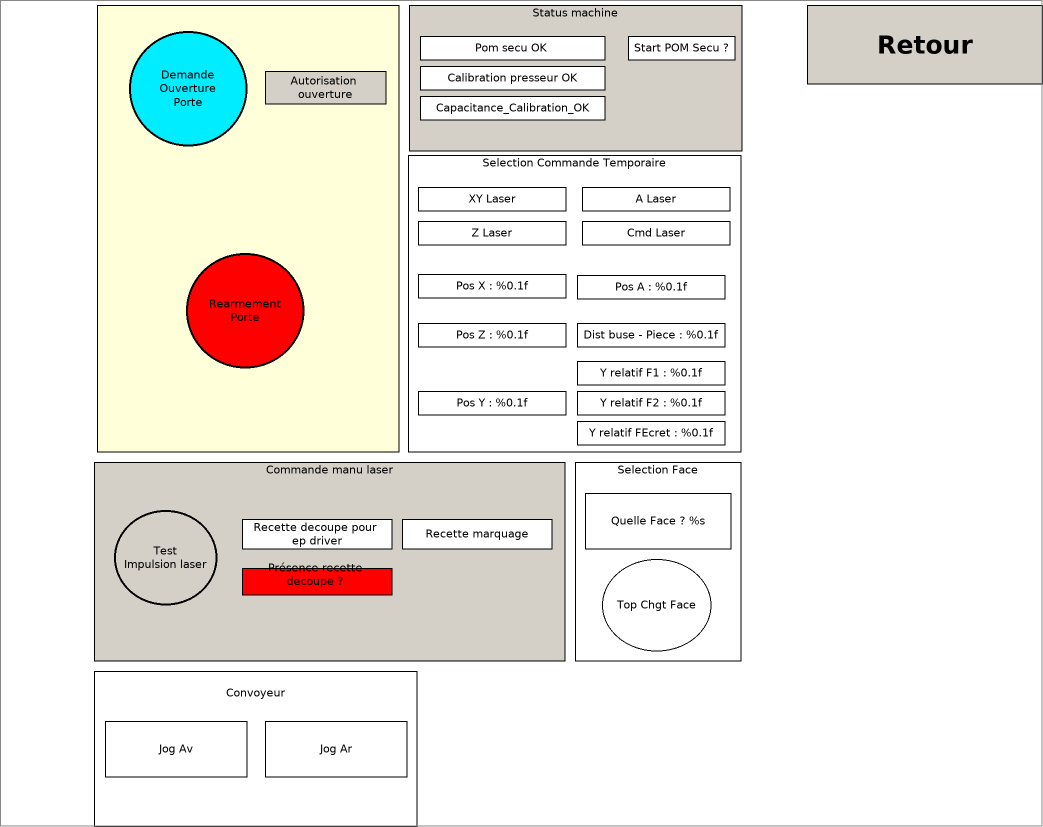
VISUALIZATION Porte_secu  // 1043x827
    Rectangle (94,462 471x199), "Commande manu laser"
    Rectangle (94,671 323x156), "Convoyeur"
        tap Gestion_ConvLaser.Jog_Av_ConvLaser
    Rectangle (97,5 302x447)
    Ellipse (129,31 118x115), "Demande Ouverture Porte", colour toggle: Attente_Arret_Propre and Clignotant_t_lent
        tap Global_Laser.Dmd_VerrDeverr_Porte
    Ellipse (186,253 118x115), "Rearmement Porte", colour toggle: RAZ_Pnoz_PorteLaser
        tap Global_Laser.Bp_Raz_Pnoz_Laser
    Rectangle (807,5 236x79), "Retour"
        OnMouseClick: change screen: Selection_Rep
        OnMouseClick: execute { Forcage_Rep.Num_Rep_Selectionne_pr_Forcage:=0; }
    RoundedRectangle (105,721 142x56), "Jog Av", colour toggle: Gestion_ConvLaser.Jog_Av_ConvLaser
        tap Gestion_ConvLaser.Jog_Av_ConvLaser
    RoundedRectangle (265,721 142x56), "Jog Ar", colour toggle: Gestion_ConvLaser.Jog_Ar_ConvLaser
        tap Gestion_ConvLaser.Jog_Ar_ConvLaser
    Rectangle (408,155 333x297), "Selection Commande Temporaire"
        tap Gestion_ConvLaser.Jog_Av_ConvLaser
    RoundedRectangle (418,187 148x24), "XY Laser", colour toggle: Selection_XYLaser
        OnMouseUp: execute {
            Selection_XYLaser :=TRUE;
            Selection_ZLaser :=FALSE;
            Selection_A		:=FALSE;
            Selection_DecManu_Laser:=false;
        }
    RoundedRectangle (418,221 148x24), "Z Laser", colour toggle: Selection_ZLaser
        OnMouseUp: execute {
            Selection_XYLaser :=FALSE;
            Selection_ZLaser :=TRUE;
            Selection_A		:=FALSE;
            Selection_DecManu_Laser :=false;
        }
    RoundedRectangle (582,187 148x24), "A Laser", colour toggle: Selection_A
        OnMouseUp: execute {
            Selection_XYLaser :=FALSE;
            Selection_ZLaser :=FALSE;
            Selection_A		:=TRUE;
        }
    Rectangle (575,462 166x199), "Selection Face"
    Ellipse (602,559 109x92), "Top Chgt Face"
        OnMouseUp: execute { top_face := TRUE; G7_Sel_Face.Test_Face:=true; }
    RoundedRectangle (585,493 146x56), "Quelle Face ? %s", text variable: Face_Cible
        OnMouseUp: write Face_Cible via VisuDialogs.Numpad, min 1, max 3
    Ellipse (114,510 103x95), "Test Impulsion laser", colour toggle: _0_LASER_ST.Dmd_Test_Tir
        tap _0_LASER_ST.Dmd_Test_Tir
    Rectangle (418,274 148x24), "Pos X : %0.1f", text variable: Pos_Reel_X_Laser
    Rectangle (418,391 148x24), "Pos Y : %0.1f", text variable: Pos_Reel_Y_Laser
    Rectangle (418,323 148x24), "Pos Z : %0.1f", text variable: Pos_Reel_Z_Laser
    Rectangle (577,275 148x24), "Pos A : %0.1f", text variable: Pos_Reel_A_Laser
    Rectangle (409,5 333x146), "Status machine"
    Rectangle (420,96 185x24), "Capacitance_Calibration_OK", colour toggle: Prog_Capacitance_Calibration_OK
    Rectangle (420,36 185x24), "Pom secu OK", colour toggle: Pom_Codeur_Secu_ok
    Rectangle (420,66 185x24), "Calibration presseur OK", colour toggle: Divers_cycles.Calib_Presseurs_OK
    RoundedRectangle (628,36 107x24), "Start POM Secu ?", colour toggle: Pom_Codeur_Secu_ok, invisible if: Pom_Codeur_Secu_ok
        OnMouseUp: execute { Divers_cycles.Step_Pom_CodeurSecu:=1; }
    Rectangle (577,361 148x24), "Y relatif F1 : %0.1f", text variable: Pos_Y_RelaFaceRef, colour toggle: Face_En_Cours <> 1
    Rectangle (577,391 148x24), "Y relatif F2 : %0.1f", text variable: Pos_Y_RelaFaceOppRef, colour toggle: Face_En_Cours <> 2
    Rectangle (577,421 148x24), "Y relatif FEcret : %0.1f", text variable: Pos_Y_RelaFaceEcret, colour toggle: Face_En_Cours <> 3
    Rectangle (577,323 148x24), "Dist buse - Piece : %0.1f", text variable: Prog_Capacitance_Actual_Value_mm, colour toggle: not Prog_Capacitance_Calibration_OK
    RoundedRectangle (242,519 150x30), "Recette decoupe pour ep driver", colour toggle: not Sel_DecMarq_Manu
        OnMouseClick: execute { Sel_DecMarq_Manu := false; }
    RoundedRectangle (402,519 150x30), "Recette marquage", colour toggle: Sel_DecMarq_Manu
        OnMouseClick: execute { Sel_DecMarq_Manu := false; }
    Rectangle (242,568 150x27), "Présence recette decoupe ?", colour toggle: Index_Recette_Decoupe <> 0
        OnMouseClick: execute { Sel_DecMarq_Manu := false; }
    RoundedRectangle (582,221 148x24), "Cmd Laser", colour toggle: Selection_DecManu_Laser
        OnMouseUp: execute {
            Selection_XYLaser :=FALSE;
            Selection_ZLaser :=FALSE;
            Selection_A		:=FALSE;
            Selection_DecManu_Laser := true;
        }
    Rectangle (265,71 121x33), "Autorisation ouverture", colour toggle: Autor_Ouverture_Porte or (Mem_Arus and Clignotant_lent)
END_VISUALIZATION

(* stored: Version 1.1.0.1
   Visu Porte_secu: Id {7749bca4-8520-4491-91db-128732bb044d} *)
